Staubli VAL3: start.pgx

program start()
begin

  taskCreate "Supervision",50,Supervision()
  taskCreate "ComPlc",50,ComPlc()
  taskCreate "Init",50,Init()

  // Mostrar pantalla d'usuari
  userPage("main")
end
